FUNCTION_BLOCK FB_MKS_903
VAR_INPUT
	stVolume : ST_Volume;
	q_xGaugeConnected	:	BOOL;
END_VAR
VAR_OUTPUT
END_VAR
VAR_IN_OUT
	stGauge	:	ST_MKS_903;
END_VAR
VAR
END_VAR

(* 
MKS 909 Vacuum gauge

A vacuum gauge takes as input, the pressure of the volume it is attached to,
and produces on its analog output, a corresponding voltage.


*)

(* Operation 
When the HV on signal is active, the gauge will take a little bit of time to
start an ion current.
*)
stGauge.tonIC.IN	:=	stGauge.i_xHvOn;	
stGauge.tonIC();

IF stGauge.tonIC.Q AND q_xGaugeConnected THEN
	stGauge.rPress := stVolume.rPressure;
	stGauge.q_iRawPress := M_MKS_903(stGauge);// gauge on
ELSIF stGauge.i_xHvOn AND q_xGaugeConnected THEN
	stGauge.rPress := 0;
	stGauge.q_iRawPress := M_MKS_903(1E-11); // gauge on, waiting for spark??
ELSE
	stGauge.rPress := 0;
	stGauge.q_iRawPress := M_MKS_903(1E-4); // gauge not on??
END_IF

METHOD PRIVATE M_MKS_903 : INT
VAR_INPUT
	stGauge	: ST_MKS_903;
END_VAR
(*
MKS 907 voltage calculation 

Does the inverse of the FB 903 from the vacuum library

A. Pai, 2017-1-13
*)
IF stGauge.rPress <> 0 THEN
	M_MKS_903 := REAL_TO_INT( (32767/10) * (LOG( stGauge.rPress ) + 11) );
ELSE
	M_MKS_903 := 0;
END_IF
END_METHOD

END_FUNCTION_BLOCK

(* stored: Version 1.1.0.1, ProductVersion 3.1.4020.12
   POU FB_MKS_903: Id {e582a674-b22f-4b02-9f19-8dbcc2feec6a}, SpecialFunc None
   Method M_MKS_903: Id {6da8ed67-5774-41ff-987a-e6754f6ebe1c} *)
